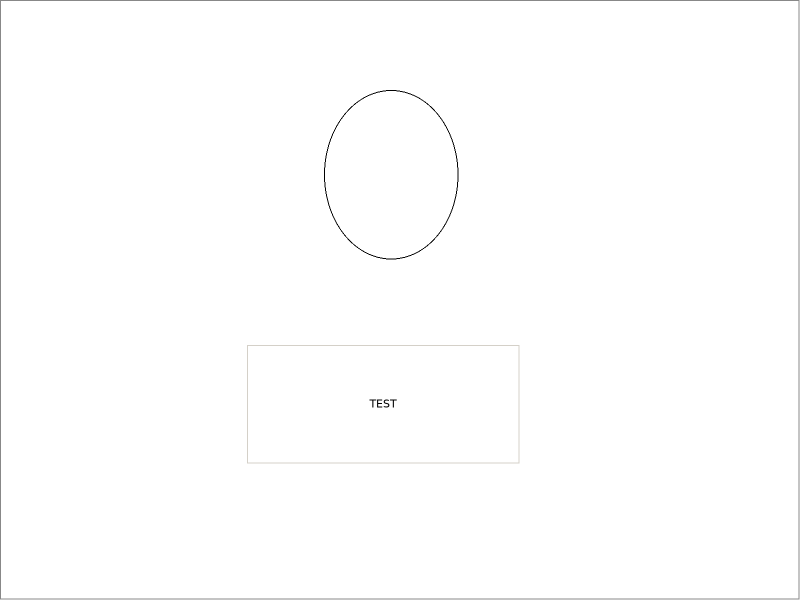
VISUALIZATION Visualization  // 800x600
    Ellipse (324,90 134x169)
    Textfield (247,345 272x118), "TEST"
END_VISUALIZATION

(* stored: Version 1.1.0.1, ProductVersion 3.1.4024.12
   Visu Visualization: Id {b308c1be-4c09-48e0-884f-39e258fee5fa} *)
